FUNCTION_BLOCK Pulse
VAR_INPUT
	enable		:	BOOL;
	offTime		:	TIME;
	onTime		:	TIME;
END_VAR
VAR_OUTPUT
	Q			:	BOOL;
END_VAR
VAR
	onTimer		:	TON;
	offTimer	:	TON;
END_VAR

offTimer(IN:= enable AND NOT(onTimer.Q), PT:= offTime, Q=> Q, ET=> );

onTimer(IN:= offTimer.Q, PT:= onTime, Q=> , ET=> );

END_FUNCTION_BLOCK

(* stored: Version 1.1.0.1, ProductVersion 3.1.4024.12
   POU Pulse: Id {82159c39-b0ea-4603-a509-8714d4a02252}, SpecialFunc None *)
